PROGRAM MAIN
VAR
	sFilePathName	: STRING := 'C:\TwinCAT\CNC\TestNci1.txt';
	sErrorMessage	: STRING := '';
	bOpen			: BOOL;
	bClose 			: BOOL;
	bSave 			: BOOL;
	bNew			: BOOL;
	nErrorCode		: USINT;
	nLineNumber		: USINT;
	bEnable: BOOL;
END_VAR



sErrorMessage	:= VisuFctTextEditorGetErrorText(usiErrCode := nErrorCode);

PRG_NcControl();
//PRG_MFuncControl();
PRG_Kinematic();

//PRG_Process();

//PRG_OpcUA();

//POU_VisButton();
POU_Process_Deneme();


	PRG_Kinematic.bExecuteKinConfigGroup;
	
	
	stAxisX.In.fSetPos;
	stAxisY.In.fSetPos;
	stAxisZ.In.fSetPos;

	
	stAxisX.In.xMove;
	stAxisY.In.xMove;
	stAxisZ.In.xMove;



AxisM1PosValue	:=	LMOD(AxisM1_B.NcToPlc.ModuloActPos,360);
AxisM2PosValue	:=	LMOD(AxisM2_C.NcToPlc.ModuloActPos,360);
AxisM3PosValue	:=	LMOD(AxisM3_A.NcToPlc.ModuloActPos,360);



	
	
	AxisXVal	:=	AxisX.NcToPlc.ActPos;
	AxisYVal	:=	AxisY.NcToPlc.ActPos;
	AxisZVal	:=	AxisZ.NcToPlc.ActPos;

END_PROGRAM

(* stored: Version 1.1.0.1, ProductVersion 3.1.4024.0
   POU MAIN: Id {2020bd6b-90a0-4fc7-9a1c-76bd8c902114}, SpecialFunc None *)
